FUNCTION_BLOCK Test_ErrorIdToString EXTENDS T_UnitTestBase
VAR_INPUT
END_VAR
VAR_OUTPUT
END_VAR
VAR
END_VAR

Assertion.AssertEquals_STRING(Expected     := 'Error 0x000012BD',
                              Actual       := F_ErrorIdToString(16#12BD),
                              VariableName := 'F_ErrorIdToString(16#12BD)');

Assertion.AssertEquals_STRING(Expected     := 'Error 0x000000FF',
                              Actual       := F_ErrorIdToString(16#FF),
                              VariableName := 'F_ErrorIdToString(16#FF)');

Assertion.AssertEquals_STRING(Expected     := 'Error 0x00000011',
                              Actual       := F_ErrorIdToString(16#11),
                              VariableName := 'F_ErrorIdToString(16#11)');

TestFinished();

END_FUNCTION_BLOCK

(* stored: Version 1.1.0.1, ProductVersion 3.1.4024.9
   POU Test_ErrorIdToString: Id {ae965cb6-9e2e-468f-834f-a33cad0a304a}, SpecialFunc None *)
